ABB RAPID module: traj1smoothed.MOD

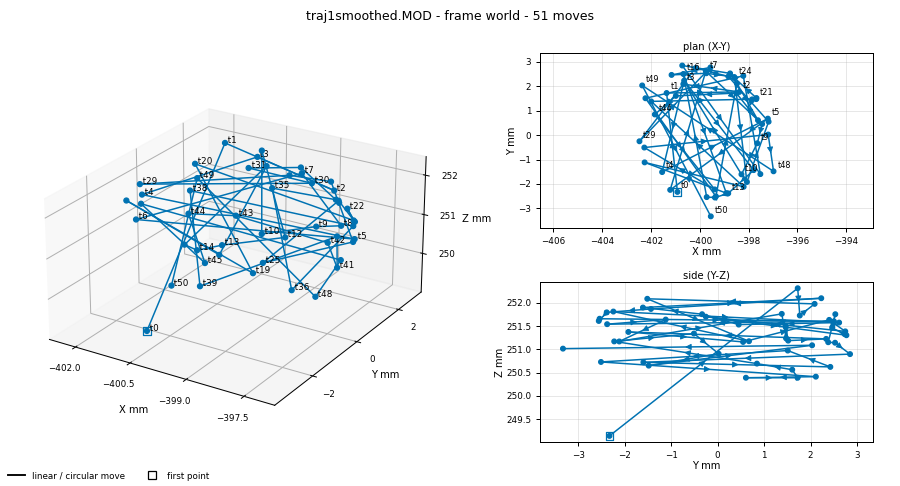
[picture p0: tool path of traj1smoothed.MOD in frame world, 51 of 52 moves have a stored position in this frame; points joined in program order, loops and branches not executed]
MODULE MainModule
PERS tooldata Servo:=[TRUE,[[0,0,114.2],[1,0,0,0]],[0.215,[8.7,12.3,49.2],[1,0,0,0],0.00021,0.00024,0.00009]];
PERS tooldata tObject:=[TRUE,[[0,0,130],[0.707106781,-0.707106781,0,0]],[0.215,[8.7,12.3,49.2],[1,0,0,0],0.00021,0.00024,0.00009]];
PERS wobjdata handpos:= [FALSE,TRUE,"",[[-400,0,250],[1,0,0,0]],[[0,0,0],[1,0,0,0]]];
    PROC main()
        ConfL\Off;
        SingArea\Wrist;
        !Startpos
        MoveAbsJ [[0.441359,-16.418,10.8814,2.79121,60.2034,-14.3875],[168.362,9E+09,9E+09,9E+09,9E+09,9E+09]] \NoEOffs, v1000, fine, wi_tGripper;
        path;
    ENDPROC
    PROC path()

VAR robtarget t0 := [[-0.9181689906476735, -2.3263351328590427, -0.8608007947843366], [0, -1, 0, 0], [0,0,-1,4], [-96,9E+09,9E+09,9E+09,9E+09,9E+09]];
VAR robtarget t1 := [[-1.3601237718987345, 1.7244733972515374, 2.316677427331113], [0, -1, 0, 0], [0,0,-1,4], [-96,9E+09,9E+09,9E+09,9E+09,9E+09]];
VAR robtarget t2 := [[1.6168640942720538, 1.7695308191693677, 1.7302847868769087], [0, -1, 0, 0], [0,0,-1,4], [-96,9E+09,9E+09,9E+09,9E+09,9E+09]];
VAR robtarget t3 := [[-0.676778467074131, 2.0886000517438643, 1.9805142987087163], [0, -1, 0, 0], [0,0,-1,4], [-96,9E+09,9E+09,9E+09,9E+09,9E+09]];
VAR robtarget t4 := [[-1.5435871188981698, -1.5129442653035898, 2.0899057931045606], [0, -1, 0, 0], [0,0,-1,4], [-96,9E+09,9E+09,9E+09,9E+09,9E+09]];
VAR robtarget t5 := [[2.785729419837538, 0.6758319691822948, 1.1766045069276834], [0, -1, 0, 0], [0,0,-1,4], [-96,9E+09,9E+09,9E+09,9E+09,9E+09]];
VAR robtarget t6 := [[-1.2138274422190538, -2.2428651618368085, 1.8153275353621146], [0, -1, 0, 0], [0,0,-1,4], [-96,9E+09,9E+09,9E+09,9E+09,9E+09]];
VAR robtarget t7 := [[0.2468689108671296, 2.6162909591654957, 1.5776996751047418], [0, -1, 0, 0], [0,0,-1,4], [-96,9E+09,9E+09,9E+09,9E+09,9E+09]];
VAR robtarget t8 := [[2.5521789782212654, 0.45428230729872865, 1.5347669071139687], [0, -1, 0, 0], [0,0,-1,4], [-96,9E+09,9E+09,9E+09,9E+09,9E+09]];
VAR robtarget t9 := [[2.3544274862083663, -0.33343754137171666, 1.7582219395113041], [0, -1, 0, 0], [0,0,-1,4], [-96,9E+09,9E+09,9E+09,9E+09,9E+09]];
VAR robtarget t10 := [[1.7054508729040174, -1.6064644884406316, 1.9018163704824853], [0, -1, 0, 0], [0,0,-1,4], [-96,9E+09,9E+09,9E+09,9E+09,9E+09]];
VAR robtarget t11 := [[-0.6422441670615004, 2.2315791815276262, 2.1019156213441694], [0, -1, 0, 0], [0,0,-1,4], [-96,9E+09,9E+09,9E+09,9E+09,9E+09]];
VAR robtarget t12 := [[2.205495323703718, -1.4340567126147468, 1.8710695810637317], [0, -1, 0, 0], [0,0,-1,4], [-96,9E+09,9E+09,9E+09,9E+09,9E+09]];
VAR robtarget t13 := [[1.1640271110855178, -2.3854119959836786, 1.7975969104796337], [0, -1, 0, 0], [0,0,-1,4], [-96,9E+09,9E+09,9E+09,9E+09,9E+09]];
VAR robtarget t14 := [[0.621216052607695, -2.5570010157722827, 1.6128604650429514], [0, -1, 0, 0], [0,0,-1,4], [-96,9E+09,9E+09,9E+09,9E+09,9E+09]];
VAR robtarget t15 := [[0.28200205062773365, -2.5389430143607417, 1.6604997657897287], [0, -1, 0, 0], [0,0,-1,4], [-96,9E+09,9E+09,9E+09,9E+09,9E+09]];
VAR robtarget t16 := [[-0.6737592819850322, 2.5045965098724325, 1.6046852830225005], [0, -1, 0, 0], [0,0,-1,4], [-96,9E+09,9E+09,9E+09,9E+09,9E+09]];
VAR robtarget t17 := [[1.086536666145088, -2.3771379829131423, 1.5433786557430627], [0, -1, 0, 0], [0,0,-1,4], [-96,9E+09,9E+09,9E+09,9E+09,9E+09]];
VAR robtarget t18 := [[-2.2616556865465203, -1.1166901433571772, 1.642823399792157], [0, -1, 0, 0], [0,0,-1,4], [-96,9E+09,9E+09,9E+09,9E+09,9E+09]];
VAR robtarget t19 := [[1.7955078022781552, -2.116017358115205, 1.1712884287282685], [0, -1, 0, 0], [0,0,-1,4], [-96,9E+09,9E+09,9E+09,9E+09,9E+09]];
VAR robtarget t20 := [[-1.9922748292469499, 1.381642591308253, 1.7652807134097994], [0, -1, 0, 0], [0,0,-1,4], [-96,9E+09,9E+09,9E+09,9E+09,9E+09]];
VAR robtarget t21 := [[2.3106682667641456, 1.4752149064215105, 1.2375978012065214], [0, -1, 0, 0], [0,0,-1,4], [-96,9E+09,9E+09,9E+09,9E+09,9E+09]];
VAR robtarget t22 := [[2.143983208989922, 1.4653234588906927, 1.4999364865010865], [0, -1, 0, 0], [0,0,-1,4], [-96,9E+09,9E+09,9E+09,9E+09,9E+09]];
VAR robtarget t23 := [[2.3195176603980974, 1.5197156200015645, 1.1892030420662563], [0, -1, 0, 0], [0,0,-1,4], [-96,9E+09,9E+09,9E+09,9E+09,9E+09]];
VAR robtarget t24 := [[1.4223268377830172, 2.3369775788573373, 1.2270551636366587], [0, -1, 0, 0], [0,0,-1,4], [-96,9E+09,9E+09,9E+09,9E+09,9E+09]];
VAR robtarget t25 := [[1.9287153095339913, -1.9196974525656312, 1.376153423661755], [0, -1, 0, 0], [0,0,-1,4], [-96,9E+09,9E+09,9E+09,9E+09,9E+09]];
VAR robtarget t26 := [[2.8171621145780437, 0.5492533223337546, 1.1614629446375695], [0, -1, 0, 0], [0,0,-1,4], [-96,9E+09,9E+09,9E+09,9E+09,9E+09]];
VAR robtarget t27 := [[1.1693671909289465, 2.4022927613869633, 1.635843726421176], [0, -1, 0, 0], [0,0,-1,4], [-96,9E+09,9E+09,9E+09,9E+09,9E+09]];
VAR robtarget t28 := [[-0.17449448699957293, 2.7486727263636475, 1.3883776395933325], [0, -1, 0, 0], [0,0,-1,4], [-96,9E+09,9E+09,9E+09,9E+09,9E+09]];
VAR robtarget t29 := [[-2.4727189452219376, -0.25253968419269945, 1.7045486524474716], [0, -1, 0, 0], [0,0,-1,4], [-96,9E+09,9E+09,9E+09,9E+09,9E+09]];
VAR robtarget t30 := [[0.43562867411655126, 2.772867131377243, 1.3054796338193349], [0, -1, 0, 0], [0,0,-1,4], [-96,9E+09,9E+09,9E+09,9E+09,9E+09]];
VAR robtarget t31 := [[-1.15791832810168, 2.466395630334971, 1.4636182180952937], [0, -1, 0, 0], [0,0,-1,4], [-96,9E+09,9E+09,9E+09,9E+09,9E+09]];
VAR robtarget t32 := [[0.2647763519670364, 2.533877328249575, 1.7579882266672184], [0, -1, 0, 0], [0,0,-1,4], [-96,9E+09,9E+09,9E+09,9E+09,9E+09]];
VAR robtarget t33 := [[1.4118810787724707, 2.3809202863159062, 1.1548383755974885], [0, -1, 0, 0], [0,0,-1,4], [-96,9E+09,9E+09,9E+09,9E+09,9E+09]];
VAR robtarget t34 := [[1.2394124382395622, 2.5285369253287553, 1.14402762177204], [0, -1, 0, 0], [0,0,-1,4], [-96,9E+09,9E+09,9E+09,9E+09,9E+09]];
VAR robtarget t35 := [[-0.7198910513402488, 2.850808125752789, 0.8992248719631879], [0, -1, 0, 0], [0,0,-1,4], [-96,9E+09,9E+09,9E+09,9E+09,9E+09]];
VAR robtarget t36 := [[2.4794955316737943, -1.5966585759850955, 0.7228523484544475], [0, -1, 0, 0], [0,0,-1,4], [-96,9E+09,9E+09,9E+09,9E+09,9E+09]];
VAR robtarget t37 := [[1.780766621314979, 2.426859589739465, 0.6238982085837566], [0, -1, 0, 0], [0,0,-1,4], [-96,9E+09,9E+09,9E+09,9E+09,9E+09]];
VAR robtarget t38 := [[-2.22791087975602, 1.5104013549192559, 0.9756826731034189], [0, -1, 0, 0], [0,0,-1,4], [-96,9E+09,9E+09,9E+09,9E+09,9E+09]];
VAR robtarget t39 := [[0.6598602346434064, -2.5092914077480253, 0.7305243891773155], [0, -1, 0, 0], [0,0,-1,4], [-96,9E+09,9E+09,9E+09,9E+09,9E+09]];
VAR robtarget t40 := [[1.5216750216995332, 2.1150106669927276, 0.41372966366463904], [0, -1, 0, 0], [0,0,-1,4], [-96,9E+09,9E+09,9E+09,9E+09,9E+09]];
VAR robtarget t41 := [[2.382497639618733, 0.6097953045866673, 0.39076212661697013], [0, -1, 0, 0], [0,0,-1,4], [-96,9E+09,9E+09,9E+09,9E+09,9E+09]];
VAR robtarget t42 := [[1.4938972243150135, 1.7223288438346227, 0.390048224604485], [0, -1, 0, 0], [0,0,-1,4], [-96,9E+09,9E+09,9E+09,9E+09,9E+09]];
VAR robtarget t43 := [[-0.982376015079537, 1.606922155382247, 0.5632306376804619], [0, -1, 0, 0], [0,0,-1,4], [-96,9E+09,9E+09,9E+09,9E+09,9E+09]];
VAR robtarget t44 := [[-1.8425359849911316, 0.8468811271802159, 0.6948977135371757], [0, -1, 0, 0], [0,0,-1,4], [-96,9E+09,9E+09,9E+09,9E+09,9E+09]];
VAR robtarget t45 := [[0.6103684141877085, -2.2244477843804926, 1.1725695658713615], [0, -1, 0, 0], [0,0,-1,4], [-96,9E+09,9E+09,9E+09,9E+09,9E+09]];
VAR robtarget t46 := [[-2.2732981136835058, -0.5088856979479146, 1.3416613221220814], [0, -1, 0, 0], [0,0,-1,4], [-96,9E+09,9E+09,9E+09,9E+09,9E+09]];
VAR robtarget t47 := [[2.8011473707645846, 0.023072555586237442, 0.9071727944755882], [0, -1, 0, 0], [0,0,-1,4], [-96,9E+09,9E+09,9E+09,9E+09,9E+09]];
VAR robtarget t48 := [[3.019451501296889, -1.4822968200293585, 0.6512665100301064], [0, -1, 0, 0], [0,0,-1,4], [-96,9E+09,9E+09,9E+09,9E+09,9E+09]];
VAR robtarget t49 := [[-2.360436807002923, 2.034553895908208, 1.0894981941530262], [0, -1, 0, 0], [0,0,-1,4], [-96,9E+09,9E+09,9E+09,9E+09,9E+09]];
VAR robtarget t50 := [[0.4495596954230223, -3.3276337578070394, 1.0171753987758925], [0, -1, 0, 0], [0,0,-1,4], [-96,9E+09,9E+09,9E+09,9E+09,9E+09]];MoveL t0, v100\V:=100.000, z1, wi_tGripper, \WObj:=handpos;
MoveL t1, v100\V:=100.000, z1, wi_tGripper, \WObj:=handpos;
MoveL t2, v100\V:=100.000, z1, wi_tGripper, \WObj:=handpos;
MoveL t3, v100\V:=100.000, z1, wi_tGripper, \WObj:=handpos;
MoveL t4, v100\V:=100.000, z1, wi_tGripper, \WObj:=handpos;
MoveL t5, v100\V:=100.000, z1, wi_tGripper, \WObj:=handpos;
MoveL t6, v100\V:=100.000, z1, wi_tGripper, \WObj:=handpos;
MoveL t7, v100\V:=100.000, z1, wi_tGripper, \WObj:=handpos;
MoveL t8, v100\V:=100.000, z1, wi_tGripper, \WObj:=handpos;
MoveL t9, v100\V:=100.000, z1, wi_tGripper, \WObj:=handpos;
MoveL t10, v100\V:=100.000, z1, wi_tGripper, \WObj:=handpos;
MoveL t11, v100\V:=100.000, z1, wi_tGripper, \WObj:=handpos;
MoveL t12, v100\V:=100.000, z1, wi_tGripper, \WObj:=handpos;
MoveL t13, v100\V:=100.000, z1, wi_tGripper, \WObj:=handpos;
MoveL t14, v100\V:=100.000, z1, wi_tGripper, \WObj:=handpos;
MoveL t15, v100\V:=100.000, z1, wi_tGripper, \WObj:=handpos;
MoveL t16, v100\V:=100.000, z1, wi_tGripper, \WObj:=handpos;
MoveL t17, v100\V:=100.000, z1, wi_tGripper, \WObj:=handpos;
MoveL t18, v100\V:=100.000, z1, wi_tGripper, \WObj:=handpos;
MoveL t19, v100\V:=100.000, z1, wi_tGripper, \WObj:=handpos;
MoveL t20, v100\V:=100.000, z1, wi_tGripper, \WObj:=handpos;
MoveL t21, v100\V:=100.000, z1, wi_tGripper, \WObj:=handpos;
MoveL t22, v100\V:=100.000, z1, wi_tGripper, \WObj:=handpos;
MoveL t23, v100\V:=100.000, z1, wi_tGripper, \WObj:=handpos;
MoveL t24, v100\V:=100.000, z1, wi_tGripper, \WObj:=handpos;
MoveL t25, v100\V:=100.000, z1, wi_tGripper, \WObj:=handpos;
MoveL t26, v100\V:=100.000, z1, wi_tGripper, \WObj:=handpos;
MoveL t27, v100\V:=100.000, z1, wi_tGripper, \WObj:=handpos;
MoveL t28, v100\V:=100.000, z1, wi_tGripper, \WObj:=handpos;
MoveL t29, v100\V:=100.000, z1, wi_tGripper, \WObj:=handpos;
MoveL t30, v100\V:=100.000, z1, wi_tGripper, \WObj:=handpos;
MoveL t31, v100\V:=100.000, z1, wi_tGripper, \WObj:=handpos;
MoveL t32, v100\V:=100.000, z1, wi_tGripper, \WObj:=handpos;
MoveL t33, v100\V:=100.000, z1, wi_tGripper, \WObj:=handpos;
MoveL t34, v100\V:=100.000, z1, wi_tGripper, \WObj:=handpos;
MoveL t35, v100\V:=100.000, z1, wi_tGripper, \WObj:=handpos;
MoveL t36, v100\V:=100.000, z1, wi_tGripper, \WObj:=handpos;
MoveL t37, v100\V:=100.000, z1, wi_tGripper, \WObj:=handpos;
MoveL t38, v100\V:=100.000, z1, wi_tGripper, \WObj:=handpos;
MoveL t39, v100\V:=100.000, z1, wi_tGripper, \WObj:=handpos;
MoveL t40, v100\V:=100.000, z1, wi_tGripper, \WObj:=handpos;
MoveL t41, v100\V:=100.000, z1, wi_tGripper, \WObj:=handpos;
MoveL t42, v100\V:=100.000, z1, wi_tGripper, \WObj:=handpos;
MoveL t43, v100\V:=100.000, z1, wi_tGripper, \WObj:=handpos;
MoveL t44, v100\V:=100.000, z1, wi_tGripper, \WObj:=handpos;
MoveL t45, v100\V:=100.000, z1, wi_tGripper, \WObj:=handpos;
MoveL t46, v100\V:=100.000, z1, wi_tGripper, \WObj:=handpos;
MoveL t47, v100\V:=100.000, z1, wi_tGripper, \WObj:=handpos;
MoveL t48, v100\V:=100.000, z1, wi_tGripper, \WObj:=handpos;
MoveL t49, v100\V:=100.000, z1, wi_tGripper, \WObj:=handpos;
MoveL t50, v100\V:=100.000, z1, wi_tGripper, \WObj:=handpos;

ENDPROC
ENDMODULE
